PROGRAM FB_TCP
VAR
END_VAR
VAR // added by the converter: edge detectors and wires of the graphical bodies
    _w1 : BOOL;
END_VAR

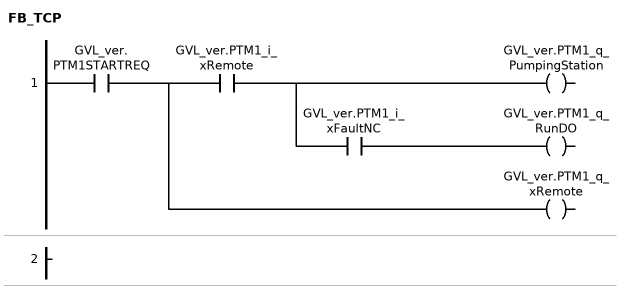
// NETWORK 1
_w1 := GVL_ver.PTM1STARTREQ AND GVL_ver.PTM1_i_xRemote;
GVL_ver.PTM1_q_PumpingStation := _w1;
GVL_ver.PTM1_q_RunDO := _w1 AND GVL_ver.PTM1_i_xFaultNC;
GVL_ver.PTM1_q_xRemote := GVL_ver.PTM1STARTREQ;

// NETWORK 2

END_PROGRAM

(* stored: Version 1.1.0.1, ProductVersion 3.1.4022.3
   POU FB_TCP: Id {46953640-11f6-42fc-9d69-f326211d57f8}, SpecialFunc None *)
